// TIA Portal V17 export
// export: Created 2026-04-13T11:12:43.4155725Z, ExportSetting WithDefaults, DisplayName Totally Integrated Automation Portal, DisplayVersion V17 Update 4, DisplayName TIA Portal Openness, DisplayVersion V17 Update 4, DisplayName TIA Portal Version Control Interface, DisplayVersion V17, DisplayName SINAMICS Startdrive Advanced, DisplayVersion V17, DisplayName SINAMICS Startdrive G130, G150, S120, S150, SINAMICS MV, S210, DisplayVersion V17, DisplayName SINAMICS Startdrive G110M, G120, G120C, G120D, G120P, G115D, DisplayVersion V17, DisplayName STEP 7 Professional, DisplayVersion V17 Update 4, DisplayName STEP 7 Safety, DisplayVersion V17, DisplayName WinCC Professional, DisplayVersion V17 Update 4
FUNCTION_BLOCK "A14-阀反馈报警"   // FB20, SCL
{ S7_Optimized_Access := 'TRUE' }
VERSION : 0.1
// stored: AutoNumber true, IsIECCheckEnabled false, IsRetainMemResEnabled false, MemoryReserve 100, SetENOAutomatically false, UDAEnableTagReadback false
   VAR
      补氮阀 : "A8-阀开关报警";
      进氮阀 : "A8-阀开关报警";
      泄压阀 : "A8-阀开关报警";
      气流雾化阀 : "A8-阀开关报警";
      输送进风阀 : "A8-阀开关报警";
      开式排风隔断阀 : "A8-阀开关报警";
      闭式排风隔断阀 : "A8-阀开关报警";
      开式进风隔断阀 : "A8-阀开关报警";
      闭式进风隔断阀 : "A8-阀开关报警";
      一级冷却水阀 : "A8-阀开关报警";
      二级冷冻水阀 : "A8-阀开关报警";
      一级排液阀 : "A8-阀开关报警";
      二级排液阀 : "A8-阀开关报警";
      除雾排液阀 : "A8-阀开关报警";
      溶剂回收排放阀 : "A8-阀开关报警";
      进风冷却水阀 : "A8-阀开关报警";
      塔顶清洗球阀 : "A8-阀开关报警";
      清洗伸缩气缸 : "A8-阀开关报警";
      "71阀开关报警_Instance" { S7_SetPoint := 'True'} : "A8-阀开关报警";
      "71阀开关报警_Instance_1" { S7_SetPoint := 'True'} : "A8-阀开关报警";
   END_VAR
BEGIN

   #补氮阀(阀开报警 => "ABD补氮阀开报警",
        阀关报警 => "ABD补氮阀关报警",
        阀状态 :="QBD补氮阀",
        阀开信号 := "IBD补氮阀开反馈",
        阀关信号 := "IBD补氮阀关反馈");

   #进氮阀(阀开报警 => "AJD进氮阀开报警",
        阀关报警 => "AJD进氮阀关报警",
        阀状态 := "QJD进氮阀",
        阀开信号 := "IJD进氮阀开反馈",
        阀关信号 := "IJD进氮阀关反馈");


   #泄压阀(阀开报警 => "AXY泄压阀开报警",
        阀关报警 => "AXY泄压阀关报警",
        阀状态 := "QXY泄压阀",
        阀开信号 := "IXY泄压阀开反馈",
        阀关信号 := "IXY泄压阀关反馈");

   #气流雾化阀(阀开报警 => "AQL气流雾化阀开报警",
          阀关报警 => "AQL气流雾化阀关报警",
          阀状态 := "QQL气流雾化阀",
          阀开信号 := "IQL气流雾化阀开反馈",
          阀关信号 := "IQL气流雾化阀关反馈");

   #输送进风阀(阀开报警 => "ASS输送进风阀开报警",
          阀关报警 => "ASS输送进风阀关报警",
          阀状态 := "QSS输送进风阀",
          阀开信号 := "ISF输送进风阀开反馈",
          阀关信号 := "ISF输送进风阀关反馈");


   #开式排风隔断阀(阀开报警 => "AKS开式排风隔断阀开报警",
            阀关报警 => "AKS开式排风隔断阀关报警",
            阀状态 := "QKS开式排风隔断阀",
            阀开信号 := "IKS开式排风隔断阀开反馈",
            阀关信号 := "IKS开式排风隔断阀关反馈");

   #闭式排风隔断阀(阀开报警 => "ABS闭式排风隔断阀开报警",
            阀关报警 => "ABS闭式排风隔断阀关报警",
            阀状态 := "QBS闭式排风隔断阀",
            阀开信号 := "IBS闭式排风隔断阀开反馈",
            阀关信号 := "IBS闭式排风隔断阀关反馈");


   #开式进风隔断阀(阀开报警 => "AKS开式进风隔断阀开报警",
            阀关报警 => "AKS开式进风隔断阀关报警",
            阀状态 := "QKS开式进风隔断阀",
            阀开信号 := "IKS开式进风隔断阀开反馈",
            阀关信号 := "IKS开式进风隔断阀关反馈");

   #闭式进风隔断阀(阀开报警 => "ABS闭式进风隔断阀开报警",
            阀关报警 => "ABS闭式进风隔断阀关报警",
            阀状态 := "QBS闭式进风隔断阀",
            阀开信号 := "IBS闭式进风隔断阀开反馈",
            阀关信号 := "IBS闭式进风隔断阀关反馈");

   #一级冷却水阀(阀开报警 => "AYJ一级冷却水阀开报警",
           阀关报警 => "AYJ一级冷却水阀关报警",
           阀状态 := "QYJ一级冷却水阀",
           阀开信号 := "IYJ一级冷却水阀开反馈",
           阀关信号 := "IYJ一级冷却水阀关反馈");


   #二级冷冻水阀(阀开报警 => "AEJ二级冷冻水阀开报警",
           阀关报警 => "AEJ二级冷冻水阀关报警",
           阀状态 := "QEJ二级冷冻水阀",
           阀开信号 := "IEJ二级冷冻水阀开反馈",
           阀关信号 := "IEJ二级冷冻水阀关反馈");

   #一级排液阀(阀开报警 => "AYJ一级排液阀开报警",
          阀关报警 => "AYJ一级排液阀关报警",
          阀状态 := "QYJ一级排液阀",
          阀开信号 := "IYJ一级排液阀开反馈",
          阀关信号 := "IYJ一级排液阀关反馈");


   #二级排液阀(阀开报警 => "AEJ二级排液阀开报警",
          阀关报警 => "AEJ二级排液阀关报警",
          阀状态 := "QEJ二级排液阀",
          阀开信号 := "IEJ二级排液阀开反馈",
          阀关信号 := "IEJ二级排液阀关反馈");

   #除雾排液阀(阀开报警 => "ACW除雾排液阀开报警",
          阀关报警 => "ACW除雾排液阀关报警",
          阀状态 := "QCW除雾排液阀",
          阀开信号 := "ICW除雾排液阀开反馈",
          阀关信号 := "ICW除雾排液阀关反馈");

   #溶剂回收排放阀(阀开报警 => "ARJ溶剂回收排放阀开报警",
            阀关报警 => "ARJ溶剂回收排放阀关报警",
            阀状态 := "QRJ溶剂回收排放阀",
            阀开信号 := "IRJ溶剂回收排放阀开反馈",
            阀关信号 := "IRJ溶剂回收排放阀关反馈");


   #进风冷却水阀(阀开报警 => "AJF进风冷却水阀开报警",
           阀关报警 => "AJF进风冷却水阀关报警",
           阀状态 := "QJF进风冷却水阀",
           阀开信号 := "IJF进风冷却水阀开反馈",
           阀关信号 := "IJF进风冷却水阀关反馈");

   #塔顶清洗球阀(阀开报警 => "ATD塔顶清洗球阀开报警",
           阀关报警 => "ATD塔顶清洗球阀关报警",
           阀状态 := "QTD塔顶清洗球阀",
           阀开信号 := "ITD塔顶清洗球阀开反馈",
           阀关信号 := "ITD塔顶清洗球阀关反馈");


   (* #清洗伸缩气缸(阀开报警 => "AQX清洗伸缩气缸开报警",
           阀关报警 => "AQX清洗伸缩气缸关报警",
           阀状态 := "QQG气缸升降阀",
           阀开信号 := "IQX清洗伸缩气缸开反馈",
           阀关信号 := "IQX清洗伸缩气缸关反馈"); *)
END_FUNCTION_BLOCK
